// TIA Portal V18 export
// export: Created 2026-01-09T11:31:56.7108796Z, ExportSetting WithDefaults, DisplayName Totally Integrated Automation Portal, DisplayVersion V18 Update 5, DisplayName TIA Portal Openness, DisplayVersion V18 Update 5, DisplayName TIA Portal Teamcenter Gateway, DisplayVersion V18, DisplayName TIA Portal Version Control Interface, DisplayVersion V18, DisplayName SINAMICS Startdrive Advanced, DisplayVersion V18 SP2 Update 1, DisplayName SINAMICS Startdrive G110M, G120, G120C, G120D, G120P, G115D, DisplayVersion V18 SP2 Update 1, DisplayName SINAMICS Startdrive G130, G150, S120, S150, SINAMICS MV, S210, G220, S200, DisplayVersion V18 SP2 Update 1, DisplayName STEP 7 Professional, DisplayVersion V18 Update 5, DisplayName STEP 7 Safety, DisplayVersion V18, DisplayName WinCC Professional, DisplayVersion V18 Update 5
TagTable "CuringOven"
  ST10_PLC_GetDB_InData_Global_Beat : Bool  (PLC tag ST10_PLC_GetDB.InData.Global.Beat, CPU S71500-2PN_TP700, 100 ms)
  ST10_PLC_GetDB_InData_Global_AutoRunning : Bool  (PLC tag ST10_PLC_GetDB.InData.Global.AutoRunning, CPU S71500-2PN_TP700, 100 ms)
  ST10_PLC_GetDB_InData_Global_Alarm : Bool  (PLC tag ST10_PLC_GetDB.InData.Global.Alarm, CPU S71500-2PN_TP700, 100 ms)
  ST10_PLC_GetDB_InData_Global_SystemStandby : Bool  (PLC tag ST10_PLC_GetDB.InData.Global.SystemStandby, CPU S71500-2PN_TP700, 100 ms)
  ST10_PLC_GetDB_InData_Global_AutoMode : Bool  (PLC tag ST10_PLC_GetDB.InData.Global.AutoMode, CPU S71500-2PN_TP700, 100 ms)
  ST10_PLC_GetDB_InData_Global_ManualMode : Bool  (PLC tag ST10_PLC_GetDB.InData.Global.ManualMode, CPU S71500-2PN_TP700, 100 ms)
  ST10_PLC_GetDB_InData_Control_AskPallet : Bool  (PLC tag ST10_PLC_GetDB.InData.Control.AskPallet, CPU S71500-2PN_TP700, 100 ms)
  ST10_PLC_GetDB_InData_Control_PalletInPos : Bool  (PLC tag ST10_PLC_GetDB.InData.Control.PalletInPos, CPU S71500-2PN_TP700, 100 ms)
  ST10_PLC_GetDB_InData_Data_CurrentTemperature_1 : Int  (PLC tag ST10_PLC_GetDB.InData.Data.CurrentTemperature_1, CPU S71500-2PN_TP700, 100 ms)
  ST10_PLC_GetDB_InData_Data_CurrentTemperature_2 : Int  (PLC tag ST10_PLC_GetDB.InData.Data.CurrentTemperature_2, CPU S71500-2PN_TP700, 100 ms)
  ST10_PLC_GetDB_InData_Data_SetTemperature : Int  (PLC tag ST10_PLC_GetDB.InData.Data.SetTemperature, CPU S71500-2PN_TP700, 100 ms)
  ST10_PLC_GetDB_InData_Data_SetSolidifyTime : Int  (PLC tag ST10_PLC_GetDB.InData.Data.SetSolidifyTime, CPU S71500-2PN_TP700, 100 ms)
  ST10_PLC_GetDB_InData_Data_ActualSolidifyTime : Int  (PLC tag ST10_PLC_GetDB.InData.Data.ActualSolidifyTime, CPU S71500-2PN_TP700, 100 ms)
